{attribute 'qualified_only' := ''}
{attribute 'strict' := ''}
TYPE MC_Direction :
(
	mcPositiveDirection := 0,
	mcShortestWay := 1,
	mcNegativeDirection := 2,
	mcCurrentDirection := 3
);
END_TYPE

(* stored: Version 1.1.0.1, ProductVersion 3.1.4024.11
   DUT MC_Direction: Id {061b8da4-d606-4aed-8a16-82b8c0a1b63a} *)
